Staubli VAL3: onF5Event.pgx

program onF5Event()
begin
  // look if the bButton is enable
  if bButton[4]
    //
    call selectType()
  endIf
end
